(* IEC 61131-3 sources: CannyIEC/st/cannyiec/functions, 1 file *)

(* ---- rsignbit-RSIGNBIT.st ---- *)
(* --- Interface --- *)
FUNCTION RSIGNBIT : BIT
VAR_INPUT
    rValue : REAL;
END_VAR

(* --- Implementation --- *)
RSIGNBIT := rValue < REAL#0;
